ADAPTER RobotInterface (* Adapter Interface *)
  (* Standard: 61499-1 *)
  (* Version 1.0, 2020-03-21, Duc Do Tran, OFFIS e.V. *)
  (* Compiler header: package fb.test; *)
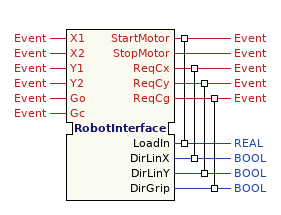
  EVENT_INPUT
    X1; (* Request from Socket *)
    X2; (* Response from Socket *)
    Y1;
    Y2;
    Go;
    Gc;
  END_EVENT
  EVENT_OUTPUT
    StartMotor WITH LoadIn; (* Indication from Plug *)
    StopMotor;
    ReqCx WITH DirLinX;
    ReqCy WITH DirLinY;
    ReqCg WITH DirGrip;
  END_EVENT
  VAR_OUTPUT
    LoadIn : REAL;
    DirLinX : BOOL;
    DirLinY : BOOL;
    DirGrip : BOOL;
  END_VAR
  SERVICE SOCKET/PLUG (* Adapter Interface *)
    SEQUENCE request_confirm
      SOCKET.REQ(REQD) -> PLUG.REQ(REQD);
      PLUG.CNF(CNFD) -> SOCKET.CNF(CNFD);
    END_SEQUENCE
    SEQUENCE indication_response
      PLUG.IND(INDD) -> SOCKET.IND(INDD);
      SOCKET.RSP(RSPD) -> PLUG.RSP(RSPD);
    END_SEQUENCE
  END_SERVICE
END_ADAPTER
